FUNCTION_BLOCK Warmlauf
VAR_INPUT
END_VAR
VAR_OUTPUT
END_VAR
VAR
	
END_VAR

END_FUNCTION_BLOCK

(* stored: Version 1.1.0.1, ProductVersion 3.1.4024.16
   POU Warmlauf: Id {324c2e16-6603-4026-8ed3-6aedaaab5116}, SpecialFunc None *)
